PROGRAM MAIN
VAR simulation : FB_SimulationBridge; lifecycle : FB_LifecycleFixture; END_VAR

simulation();
lifecycle();

END_PROGRAM

(* stored: Version 1.1.0.1
   POU MAIN: Id {36635085-d5ca-41a8-8359-e4425be93533} *)
